% RSLogix 500 project 20230719_MicroLogix_1100_driver_of_Micro8xx_2080-MOT-HSC.RSS, saved by version 8.30.00.16 %
PROJECT "UNTITLED"    % processor: Bul.1763 MicroLogix 1100 Series B %

PROGRAM FILES
  LAD 2   3 rungs

DATA FILES
  O0 OUTPUT  4 elements
  I1 INPUT  6 elements
  S2 STATUS  66 elements
  B3 BINARY  1 elements
  T4 TIMER  4 elements
  C5 COUNTER  1 elements
  R6 CONTROL  1 elements
  N7 INTEGER  1 elements
  F8 FLOAT  1 elements

LADDER 2
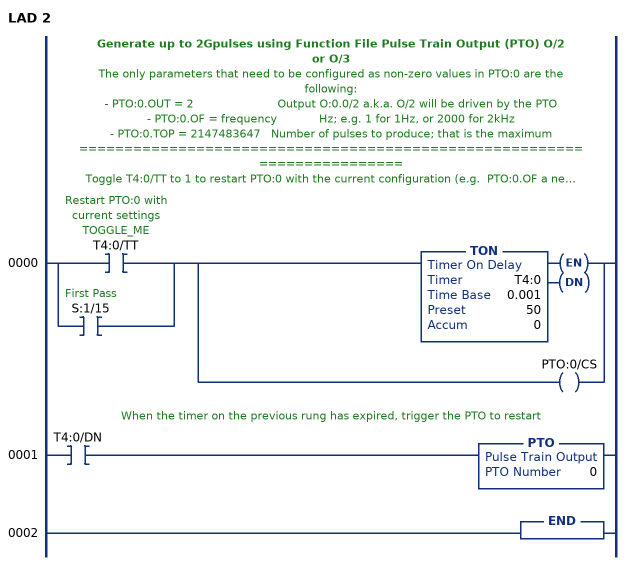
% Rung: 0 %
% TITLE: Generate up to 2Gpulses using Function File Pulse Train Output (PTO) O/2 or O/3 %
% The only parameters that need to be configured as non-zero values in PTO:0 are the following:
% - PTO:0.OUT = 2                        Output O:0.0/2 a.k.a. O/2 will be driven by the PTO
% - PTO:0.OF = frequency            Hz; e.g. 1 for 1Hz, or 2000 for 2kHz
% - PTO:0.TOP = 2147483647   Number of pulses to produce; that is the maximum
% ========================================================================
% 
% Toggle T4:0/TT to 1 to restart PTO:0 with the current configuration (e.g.  PTO:0.OF a new output frequency)
% - Start a 50ms timer, which will reset when it expires
% - PTO:0.CS (Control Stop) will  become 1 at first, then 0 when the timer expires %
SOR BST XIC T4:0/TT NXB XIC S:1/15 BND BST TON T4:0 0.001 50 0 NXB OTE PTO:0/CS BND EOR
%   T4:0/TT  TOGGLE_ME  "Restart PTO:0 with current settings" %
%   S:1/15  "First Pass" %
% Rung: 1 %
% When the timer on the previous rung has expired, trigger the PTO to restart %
SOR XIC T4:0/DN PTO 0 EOR
% Rung: 2 %
SOR END EOR

DATA TABLE (non-zero values as saved)
DATA T4
% .PRE .ACC %
% T4:0 % 50 0
% T4:1 % 51 0
% T4:2 % 2560 0
% T4:3 % 5120 0
DATA C5
% .PRE .ACC %
% C5:0 % 6001 0
